{attribute addProperty BoxType "AT2042-0250-0024"}
{attribute addProperty Id "A_0098_AT2025_5250_0019_AT2025_5250AT2025_C5E5984862678.25"}
{attribute addProperty CRC "904647970"}
{attribute addProperty SizeInBites "626"}
{attribute addProperty SizeInBytes "78.25"}
TYPE A_0046_AT2042_0250_0024_35EBD522 EXTENDS AT2042_BA5A9548 :
STRUCT
	{attribute addProperty Name "A_0098_AT2025_5250_0019_AT2025_5250"}
	A_0098_AT2025_5250_0019_AT2025_5250 : AT2025_C5E59848;
END_STRUCT
END_TYPE

(* stored: Version 1.2.0.0, ProductVersion 3.1.4024.9
   DUT A_0046_AT2042_0250_0024_35EBD522: Id {4c6b3187-ede0-443f-b02d-a49cd5598d1e} *)
